FUNCTION_BLOCK FB_HeatpumpOperation
VAR_IN_OUT
	MBMaster		:	ModbusRtuMasterV2_KL6x22B;
	Get				:	ST_HeatpumpGet;
END_VAR

VAR_INPUT
	ACPowerStatus	:	BOOL;
	HeatPumpID		:	BYTE;
	MBFree			:	BOOL;
	OperatingPoint	:	st_OperatingPoint;
	SFCInit			:	BOOL;
END_VAR
		
VAR
	DataBuffer				:	ARRAY[0..50] OF WORD;
	b_MBBusy				:	BOOL;
	b_MBerr					:	BOOL;
	ui_cbRead				:	UINT;
	b_EnableTransmission	:	BOOL;
	ModbusStartTrigger		:	R_Trig;
	MBRetryCount			:	BYTE;
	ModbusRetryTimer		:	TON := (PT := TIME#250MS);
	ResetRetryTimer			:	Bool;
	SendValue		:	WORD;
	TransmissionDoneTrigger	:	F_Trig;
	
	ReadSetpointHeating		:	REAL;
	ReadSetpointCooling		:	REAL;
	ReadCoolingMode			:	WORD;
	Writeregstatus			:	WORD;
END_VAR

VAR_OUTPUT
	MBCommBusy				:	Bool;
END_VAR

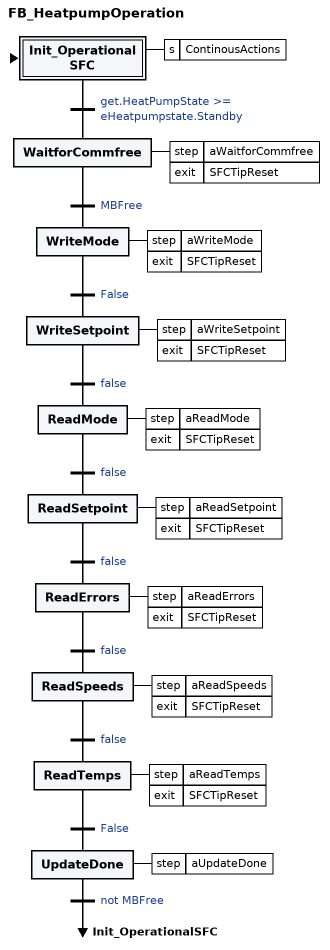
INITIAL_STEP Init_OperationalSFC:
    ContinousActions(s);
END_STEP
TRANSITION FROM Init_OperationalSFC TO WaitforCommfree
    := get.HeatPumpState >= eHeatpumpstate.Standby;
END_TRANSITION
STEP WaitforCommfree:
    aWaitforCommfree(N);  // step action
    SFCTipReset(P0);  // exit action
END_STEP
TRANSITION FROM WaitforCommfree TO WriteMode
    := MBFree;
END_TRANSITION
STEP WriteMode:
    aWriteMode(N);  // step action
    SFCTipReset(P0);  // exit action
END_STEP
TRANSITION FROM WriteMode TO WriteSetpoint
    := False;
END_TRANSITION
STEP WriteSetpoint:
    aWriteSetpoint(N);  // step action
    SFCTipReset(P0);  // exit action
END_STEP
TRANSITION FROM WriteSetpoint TO ReadMode
    := false;
END_TRANSITION
STEP ReadMode:
    aReadMode(N);  // step action
    SFCTipReset(P0);  // exit action
END_STEP
TRANSITION FROM ReadMode TO ReadSetpoint
    := false;
END_TRANSITION
STEP ReadSetpoint:
    aReadSetpoint(N);  // step action
    SFCTipReset(P0);  // exit action
END_STEP
TRANSITION FROM ReadSetpoint TO ReadErrors
    := false;
END_TRANSITION
STEP ReadErrors:
    aReadErrors(N);  // step action
    SFCTipReset(P0);  // exit action
END_STEP
TRANSITION FROM ReadErrors TO ReadSpeeds
    := false;
END_TRANSITION
STEP ReadSpeeds:
    aReadSpeeds(N);  // step action
    SFCTipReset(P0);  // exit action
END_STEP
TRANSITION FROM ReadSpeeds TO ReadTemps
    := false;
END_TRANSITION
STEP ReadTemps:
    aReadTemps(N);  // step action
    SFCTipReset(P0);  // exit action
END_STEP
TRANSITION FROM ReadTemps TO UpdateDone
    := False;
END_TRANSITION
STEP UpdateDone:
    aUpdateDone(N);  // step action
END_STEP
TRANSITION FROM UpdateDone TO Init_OperationalSFC
    := not MBFree;
END_TRANSITION

ACTION aReadErrors:

MBMaster.ReadRegs(	UnitID 		:= 	HeatPumpID,
					Quantity 	:= 	7,
					MBAddr		:=	950,
					cbLength 	:= 	7*2,
					pMemoryAddr	:=	ADR(DataBuffer),
					Execute		:=	ModbusStartTrigger.Q,
					Timeout		:=	T#250MS,		
					Busy		=>	b_MBBusy,
					Error 		=>	b_MBerr,
					cbRead 		=>	ui_cbRead
					);

TransmissionDoneTrigger(clk := b_MBBusy);

IF TransmissionDoneTrigger.q THEN
	IF NOT b_MBerr THEN
		
		ParseHeatPumpErrors(	w_Alarms1 := DataBuffer[0],
								w_Alarms2 := DataBuffer[1],
								w_Alarms3 := DataBuffer[2],
								w_Alarms4 := DataBuffer[3],
								w_Alarms5 := DataBuffer[4],
								w_Alarms6 := DataBuffer[5],
								w_Alarms7 := DataBuffer[6],
								Get := Get			
							);
		
		//done, preset for next step
		
		MBRetryCount := 0;
		sfctip := TRUE;
	ELSE
		MBRetryCount := MBRetryCount + 1;
		b_EnableTransmission	:= FALSE;
				
		//if comm fails 5 times in a row. system is unusable
		IF MBRetryCount > 5 THEN
			get.HeatPumpState := eHeatpumpState.ERROR;
			get.Events.b_CommError := TRUE;
		END_IF
	END_IF
END_IF
END_ACTION

ACTION aReadMode:

MBMaster.ReadRegs(	UnitID 		:= 	HeatPumpID,
					Quantity 	:= 	1,
					MBAddr		:=	200,
					cbLength 	:= 	10,
					pMemoryAddr	:=	ADR(DataBuffer),
					Execute		:=	ModbusStartTrigger.Q,
					Timeout		:=	T#250MS,		
					Busy		=>	b_MBBusy,
					Error 		=>	b_MBerr,
					cbRead 		=>	ui_cbRead
					);

TransmissionDoneTrigger(clk := b_MBBusy);

IF TransmissionDoneTrigger.q THEN
	IF NOT b_MBerr THEN
	
		//transmission done, process data
		CASE DataBuffer[0] OF
			0:	get.HeatPumpState := eHeatpumpState.Standby;
			1:	get.HeatPumpState := eHeatpumpState.Active_Cooling;
			2:	get.HeatPumpState := eHeatpumpState.Active_Heating;
		END_CASE
		
		//done, preset for next step
		b_EnableTransmission := FALSE;
		ModbusStartTrigger(clk := b_EnableTransmission);
		MBRetryCount := 0;
		sfctip := TRUE;
	ELSE
		MBRetryCount := MBRetryCount + 1;
		b_EnableTransmission	:= FALSE;
		
		//if comm fails 5 times in a row. system is unusable
		IF MBRetryCount > 5 THEN
			get.HeatPumpState := eHeatpumpState.ERROR;
			get.Events.b_CommError := TRUE;
		END_IF
	END_IF
END_IF
END_ACTION

ACTION aReadSetpoint:

//r_FanSpeedPCT			:	REAL;		//7000
//r_PumpSpeedPCT		:	REAL;		//7001

MBMaster.ReadRegs(	UnitID 		:= 	HeatPumpID,
					Quantity 	:= 	2,
					MBAddr		:=	7203,
					cbLength 	:= 	10,
					pMemoryAddr	:=	ADR(DataBuffer),
					Execute		:=	ModbusStartTrigger.Q,
					Timeout		:=	T#250MS,		
					Busy		=>	b_MBBusy,
					Error 		=>	b_MBerr,
					cbRead 		=>	ui_cbRead
					);

TransmissionDoneTrigger(clk := b_MBBusy);

IF TransmissionDoneTrigger.q THEN
	IF NOT b_MBerr THEN
	
		//transmission done, process data
		get.HeatpumpData.r_SetpointHeating	:=	DataBuffer[1]/10;
		get.HeatpumpData.r_SetpointCooling	:=	DataBuffer[0]/10;
			
		//done, preset for next step
		b_EnableTransmission := FALSE;
		ModbusStartTrigger(clk := b_EnableTransmission);
		MBRetryCount := 0;
		sfctip := TRUE;
	ELSE
		MBRetryCount := MBRetryCount + 1;
		b_EnableTransmission	:= FALSE;
		
		//if comm fails 5 times in a row. system is unusable
		IF MBRetryCount > 5 THEN
			get.HeatPumpState := eHeatpumpState.ERROR;
			get.Events.b_CommError := TRUE;
		END_IF
	END_IF
END_IF
END_ACTION

ACTION aReadSpeeds:

//r_FanSpeedPCT			:	REAL;		//7000
//r_PumpSpeedPCT		:	REAL;		//7001

MBMaster.ReadRegs(	UnitID 		:= 	HeatPumpID,
					Quantity 	:= 	2,
					MBAddr		:=	7000,
					cbLength 	:= 	4,
					pMemoryAddr	:=	ADR(DataBuffer),
					Execute		:=	ModbusStartTrigger.Q,
					Timeout		:=	T#250MS,		
					Busy		=>	b_MBBusy,
					Error 		=>	b_MBerr,
					cbRead 		=>	ui_cbRead
					);

TransmissionDoneTrigger(clk := b_MBBusy);

IF TransmissionDoneTrigger.q THEN
	IF NOT b_MBerr THEN
		
		//transmission done, process data
		get.HeatpumpData.r_FanSpeedPCT		:=	WORD_TO_REAL(DataBuffer[0])/10;
		get.HeatpumpData.r_PumpSpeedPCT		:= 	WORD_TO_REAL(DataBuffer[1])/10;
		
		//done, preset for next step
		b_EnableTransmission := FALSE;
		ModbusStartTrigger(clk := b_EnableTransmission);
		MBRetryCount := 0;
		sfctip := TRUE;
	ELSE
		MBRetryCount := MBRetryCount + 1;
		b_EnableTransmission	:= FALSE;
		
		//if comm fails 5 times in a row. system is unusable
		IF MBRetryCount > 5 THEN
			get.HeatPumpState := eHeatpumpState.ERROR;
			get.Events.b_CommError := TRUE;
		END_IF
	END_IF
END_IF
END_ACTION

ACTION aReadTemps:

(*
r_InletWaterTemp	:	REAL;		//400
r_OutletWaterTemp	:	REAL;		//401
r_HighPressure		:	REAL;		//406
r_LowPressure		:	REAL;		//414
r_CompInputTemp		:	REAL;		//422
r_OutdoorTemp		:	REAL;		//428
r_CompOutputTemp	:	REAL;		//433-435
ui_WaterFlowRate		:	uINT;		//444
*)

MBMaster.ReadRegs(	UnitID 		:= 	HeatPumpID,
					Quantity 	:= 	45,
					MBAddr		:=	400,
					cbLength 	:= 	90,
					pMemoryAddr	:=	ADR(DataBuffer),
					Execute		:=	ModbusStartTrigger.Q,
					Timeout		:=	T#250MS,		
					Busy		=>	b_MBBusy,
					Error 		=>	b_MBerr,
					cbRead 		=>	ui_cbRead
					);

TransmissionDoneTrigger(clk := b_MBBusy);

IF TransmissionDoneTrigger.q THEN
	IF NOT b_MBerr THEN
		
		//transmission done, process data
		get.HeatpumpData.r_InletWaterTemp		:=	WORD_TO_REAL(DataBuffer[0])/10;
		get.HeatpumpData.r_OutletWaterTemp		:= 	WORD_TO_REAL(DataBuffer[1])/10;
		get.HeatpumpData.r_HighPressure			:=	WORD_TO_REAL(DataBuffer[6])/100;
		get.HeatpumpData.r_LowPressure			:= 	WORD_TO_REAL(DataBuffer[14])/100;
		get.HeatpumpData.r_CompInputTemp		:=	WORD_TO_REAL(DataBuffer[22])/10;
		get.HeatpumpData.r_OutdoorTemp			:= 	WORD_TO_REAL(DataBuffer[28])/10;
		get.HeatpumpData.r_CompOutputTemp		:=	WORD_TO_REAL(DataBuffer[33])/10;	//comp dischyarge 1 for now
		get.HeatpumpData.ui_WaterFlowRate			:= 	DataBuffer[44];
		
		//done, preset for next step
		b_EnableTransmission := FALSE;
		ModbusStartTrigger(clk := b_EnableTransmission);
		MBRetryCount := 0;
		sfctip := TRUE;
	ELSE
		MBRetryCount := MBRetryCount + 1;
		b_EnableTransmission	:= FALSE;
		
		//if comm fails 5 times in a row. system is unusable
		IF MBRetryCount > 5 THEN
			get.HeatPumpState := eHeatpumpState.ERROR;
			get.Events.b_CommError := TRUE;
		END_IF
	END_IF
END_IF
END_ACTION

ACTION aUpdateDone:
SFCTip := FALSE;
MBCommBusy := False;
END_ACTION

ACTION aWaitforCommfree:
//SFCTip := FALSE;
//b_EnableTransmission	:= FALSE;
//ModbusStartTrigger(clk := b_EnableTransmission);
END_ACTION

ACTION aWriteMode:
//SFCTip := FALSE;


//b_EnableTransmission	:= TRUE;
//ModbusStartTrigger(clk := b_EnableTransmission);

Databuffer[0]	:= OperatingPoint.OperatingMode;	//set operating mode for write
Databuffer[1]	:= 3;								//enable write registers

MBMaster.WriteRegs ( 
					UnitID 		:= 	HeatPumpID,
					Quantity 	:= 	2,
					MBAddr		:=	7200,
					cbLength 	:= 	4,
					pMemoryAddr	:=	ADR(Databuffer),
					Execute		:=	ModbusStartTrigger.Q,
					Timeout		:=	T#250MS,		
					Busy		=>	b_MBBusy,
					Error 		=>	b_MBerr,
					);
				

TransmissionDoneTrigger(clk := b_MBBusy);

IF TransmissionDoneTrigger.q THEN
	IF NOT b_MBerr THEN
				
		//done, preset for next step
		b_EnableTransmission := FALSE;
		ModbusStartTrigger(clk := b_EnableTransmission);
		MBRetryCount := 0;
		sfctip := TRUE;
	ELSE
		MBRetryCount := MBRetryCount + 1;
		b_EnableTransmission	:= FALSE;
		
		//if comm fails 5 times in a row. system is unusable
		IF MBRetryCount > 5 THEN
			get.HeatPumpState := eHeatpumpState.ERROR;
			get.Events.b_CommError := TRUE;
		END_IF
	END_IF
END_IF
END_ACTION

ACTION aWriteSetpoint:

CASE OperatingPoint.OperatingMode OF				//Update setpoint depending on mode
	eHeatPumpMode.Cooling:
		Databuffer[0]	:= REAL_TO_WORD(LIMIT(50, ((Operatingpoint.Setpoint)*10), 230));
		Databuffer[1]	:= REAL_TO_WORD(Get.HeatpumpData.r_SetpointHeating*10);
	eHeatPumpMode.Heating:
		Databuffer[0]	:= REAL_TO_WORD(Get.HeatpumpData.r_SetpointCooling*10);
		Databuffer[1]	:= REAL_TO_WORD(LIMIT(250, ((Operatingpoint.Setpoint)*10), 550));
	eHeatPumpMode.Standby:
		Databuffer[0]	:= REAL_TO_WORD(Get.HeatpumpData.r_SetpointCooling*10);
		Databuffer[1]	:= REAL_TO_WORD(Get.HeatpumpData.r_SetpointHeating*10);	
END_CASE

MBMaster.WriteRegs (
		UnitID 		:= 	HeatPumpID,
		Quantity 	:= 	2,
		MBAddr		:=	7203,
		cbLength 	:= 	4,
		pMemoryAddr	:=	ADR(Databuffer),
		Execute		:=	ModbusStartTrigger.Q,
		Timeout		:=	T#250MS,		
		Busy		=>	b_MBBusy,
		Error 		=>	b_MBerr,
);


TransmissionDoneTrigger(clk := b_MBBusy);

IF TransmissionDoneTrigger.q THEN
	IF NOT b_MBerr THEN
		//done, preset for next step

		MBRetryCount := 0;
		sfctip := TRUE;
	ELSE
		MBRetryCount := MBRetryCount + 1;
		b_EnableTransmission	:= FALSE;
		
		//if comm fails 5 times in a row. system is unusable
		IF MBRetryCount > 5 THEN
			get.HeatPumpState := eHeatpumpState.ERROR;
			get.Events.b_CommError := TRUE;
		END_IF
	END_IF
END_IF
END_ACTION

ACTION ContinousActions:
//sfctip := False;
ModbusRetryTimer(in:= NOT (ModbusRetryTimer.Q OR ResetRetryTimer));
ModbusStartTrigger(clk := ModbusRetryTimer.q);

//for initial use, get notice if 1 packet fails
IF MBRetryCount > 1 THEN
	get.Events.b_CommWarning := TRUE;
END_IF

//ResetRetryTimer := FALSE;
END_ACTION

METHOD ParseHeatPumpErrors : BOOL
VAR_INPUT
	w_Alarms1	:	WORD;
	w_Alarms2	:	WORD;
	w_Alarms3	:	WORD;
	w_Alarms4	:	WORD;
	w_Alarms5	:	WORD;
	w_Alarms6	:	WORD;
	w_Alarms7	:	WORD;
END_VAR		
VAR
	
END_VAR

VAR_IN_OUT
	get	:	ST_HeatpumpGet;	
END_VAR
get.events.b_ProbeError		:=	WORD_TO_BOOL(w_Alarms3) OR WORD_TO_BOOL(w_Alarms4) OR w_Alarms5.0;

get.events.b_PressureError		:=	w_Alarms1.0 OR	//E001: High Pressure
									w_Alarms1.1 OR //E002: Low Pressure
									w_Alarms2.3;	//E020: Inverted Pressure Transducers


get.events.b_CompressorError	:=	w_Alarms1.2 OR //E003: Compressor overheated
									w_Alarms1.7 OR //E008: Compressor underspeed
									w_Alarms1.8 OR	//E009: High disch temp
									w_Alarms1.12 OR //E013: Comp2 Overheated
									w_Alarms2.2 OR	//E019: CP2 High disch temp
									w_Alarms2.6 OR	//E023: Comp3 Overheated
									w_Alarms5.1 OR //'E801: Link Inverter1',
									w_Alarms5.2 OR //'E802: Link Inverter2',
									w_Alarms5.3 OR //'E803: Link Inverter3',
									w_Alarms5.4 OR //'E851: HWfault Inverter1',
									w_Alarms5.5 OR //'E852: HWfault Inverter2',
									w_Alarms5.6 OR //'E853: HWfault Inverter3',
									w_Alarms5.7 OR //'E861: OverCurrent Inv1',
									w_Alarms5.8 OR //'E862: OverCurrent Inv2',
									w_Alarms5.9 OR //'E863: OverCurrent Inv3',
									w_Alarms5.10 OR //'E871: High Temp Inv1',
									w_Alarms5.11 OR //'E872: High Temp Inv2',
									w_Alarms5.12 OR //'E873: High Temp Inv3',
									w_Alarms5.13 OR //'E881: Bad Voltage Inv1',
									w_Alarms5.14 OR //'E882: Bad Voltage Inv2',
									w_Alarms5.15 OR //'E883: Bad Voltage Inv3',
									w_Alarms6.0 OR //E891: Phase Seq Inv1',
									w_Alarms6.1 OR //'E892: Phase Seq Inv2',
									w_Alarms6.2 OR //'E893: Phase Seq Inv3',
									w_Alarms6.3 OR //'E901: Model err Inv1',
									w_Alarms6.4 OR //'E902: Model err Inv2',
									w_Alarms6.5 OR //'E903: Model err Inv3',
									w_Alarms6.6 OR //'E911: Ovl error Inv1',
									w_Alarms6.7 OR //'E9112: Ovl error Inv2',
									w_Alarms6.8 OR //'E913: Ovl error Inv3',
									w_Alarms6.9 OR //'E921: Overc PFC Inv1',
									w_Alarms6.10 OR //'E922: Overc PFC Inv2',
									w_Alarms6.11 OR //'E923: Overc PFC Inv3',
									w_Alarms6.12 OR //'E931: Int Com ERR Inv1',
									w_Alarms6.13 OR //'E932: Int Com ERR Inv2',
									w_Alarms6.14 OR //'E933: Int Com ERR Inv3',
									w_Alarms6.15 OR //'E941: Fault PFC Inv1',
									w_Alarms7.0 OR //E942: Fault PFC Inv2
									w_Alarms7.1 OR //'E943: Fault PFC Inv3',
									w_Alarms7.2 OR //'E951: Probe error Inv1',
									w_Alarms7.3 OR //'E952: Probe error Inv2',
									w_Alarms7.4 OR //'E953: Probe error Inv3',
									w_Alarms7.5 OR //'E961: Abnormal Cond Inv1',
									w_Alarms7.6 OR //'E962: Abnormal Cond Inv2',
									w_Alarms7.7 OR //'E963: Abnormal Cond Inv3',
									w_Alarms7.8 OR //'E971: Inv1 Eeprom Error',
									w_Alarms7.9 OR //'E972: Inv2 Eeprom Error',
									w_Alarms7.10 OR //'E973: Inv3 Eeprom Error',
									w_Alarms7.11;	//E029: CP3 High disch temp

get.events.b_ValveError		:=		w_Alarms2.11; //E041: Incongruent temps;


get.events.b_FanError			:=	w_Alarms1.2 OR //E004: Fan Overheated	
									w_Alarms1.13 OR //E014: Fan2 Overheated 
									w_Alarms2.7;	//E024: Fan3 Overheated					

get.events.b_PumpError			:=	w_Alarms1.5 OR	 	//E006: Lack of flow
									w_Alarms1.15 OR 	//E016: Pump Overheated
									w_Alarms2.9;		//E026: Pump2 Overheated

get.events.b_WaterTempError		:=	w_Alarms2.1 OR	//E018: OverTemperature
									w_Alarms1.4;	//E005: Frost

get.events.b_IOError			:=	w_Alarms2.14 OR 	//E101: IOMod1 Disconnected
									w_Alarms2.15; 		//E102: IOMod2 Disconnected
END_METHOD

ACTION SFCTipReset:
SFCTip := FALSE;
ResetRetryTimer := FALSE;
END_ACTION

END_FUNCTION_BLOCK

(* stored: Version 1.1.0.1, ProductVersion 3.1.4024.12
   POU FB_HeatpumpOperation: Id {901aaa6c-6f92-468b-b3cb-00ad11f4a925}, SpecialFunc None
   Action aReadErrors: Id {b7820a4c-7d81-4d6c-b5a4-1d097a84603f}
   Action aReadMode: Id {3ea409e0-0dd8-4b16-8ed1-2c6e6f01e327}
   Action aReadSetpoint: Id {6b88302c-ef6e-45d7-b3e3-e541daa0bd1f}
   Action aReadSpeeds: Id {0855ff15-4f1e-44c9-8172-e09c4ea72d8c}
   Action aReadTemps: Id {5d48e278-a0db-44bc-8734-1201088798dc}
   Action aUpdateDone: Id {610d1b2f-4e5d-47c0-b950-f958ae2abc9d}
   Action aWaitforCommfree: Id {beec0e0f-8192-4b64-880b-e0e737f9b33c}
   Action aWriteMode: Id {f5867f2c-079b-4415-a7d5-dbc8b972edd0}
   Action aWriteSetpoint: Id {abf1e94c-32a9-442b-ab9d-702ccde5284d}
   Action ContinousActions: Id {46176823-239b-49e9-9712-bad7a3a146b9}
   Method ParseHeatPumpErrors: Id {70776e8e-d21c-4087-9eb3-c68344ed5cdf}
   Action SFCTipReset: Id {e088e94f-7658-429f-b3f5-865b10b699f8} *)
